(* CODESYS project tc_helper.library
   Author: R. Christopher
   Title: Tc_Helper
   Version: 1.0.0.8
   DefaultNamespace: Tc_Helper
   Company: Red Rock Controls
   Description: Clock.DateTimeInitialised added
      
      Copyright Red Rock Controls Limited 2014

Project tree, tasks and I/O mapping:
  libraries: Tc2_Standard, * (Beckhoff Automation GmbH); Tc2_System, * (Beckhoff Automation GmbH); Tc2_Utilities, * (Beckhoff Automation GmbH)
  Classes/
    function block TClock [ST]: DateAsString, DateTimeAsString, DateTimeInitialised, NowAsDateTime, NowAsTimeStruct, TimeAsString
    function block TCounter [ST]: Dec, Inc, Reset, Value, ValueAsTArg
    function block TFallingEdge [ST]: Test
    function block TOnTimer [ST]: FB_init, PresetTime, Reset, Run
    function block TRisingEdge [ST]: Test
    function block TStringSplitter [ST]: GetNext, Init
  Functions/
    function F_Concat2 [ST]
    function F_Concat4 [ST]
    function F_Concat6 [ST]
    function F_Concat8 [ST]
    function F_FormatString1 [ST]
    function F_FormatString2 [ST]
    function F_FormatString3 [ST]
    function F_FormatStringEx1 [ST]
    function F_FormatStringEx2 [ST]
    function F_FormatStringEx3 [ST]
    function F_FormatStringEx4 [ST]
    function F_LREAL_TO_STRING [ST]
    function F_LTrimEx [ST]
    function F_StripLF [ST]
    function F_Trim [ST]
    function F_UDINT_TO_STRING [ST]
  Version/
    global variables Global_Version
*)

// Version/Global_Version
// This function has been automatically generated from the project information.
VAR_GLOBAL CONSTANT
	{attribute 'const_non_replaced'}
	stLibVersion_Tc_Helper : ST_LibVersion := (iMajor := 1, iMinor := 0, iBuild := 0, iRevision := 8, sVersion := '1.0.0.8');
END_VAR

// Classes/TClock
FUNCTION_BLOCK TClock
VAR
    _DateTimeInitialised : BOOL; // to detect startup
	_NowAsTimeStruct: TIMESTRUCT;
    
	NT_GetTime1: NT_GetTime;
	TON1: TON;
    GetWindowsTimeRequest : BOOL;
	SyncRequest: BOOL;
    F_TRIG1 : F_TRIG;
	RTC_EX2: RTC_EX2;
	PresetTime: TIMESTRUCT;
END_VAR

// Request a sync every 10s
TON1(IN := NOT GetWindowsTimeRequest, PT := T#10S, Q=> GetWindowsTimeRequest);

// Get time from Windows clock
NT_GetTime1(
	NetId := '',
	Start := GetWindowsTimeRequest OR NOT _DateTimeInitialised, // request on first scan also
	TmOut := T#2S,
    Busy => ,
    Err => ,
    ErrId => ,
	TimeStr => PresetTime);

// Request sync to Windows time when time received
F_TRIG1(CLK :=  NT_GetTime1.Busy, Q=> SyncRequest);   
    
// Sync RTC to Windows time
RTC_EX2(
	EN:= SyncRequest, // re-initialise to Windows clock following sync request
	PDT:= PresetTime, // time to sync to
	PMICRO:= PresetTime.wMilliseconds, 
	Q=> , 
	CDT=> _NowAsTimeStruct, // time updated on every call
	CMICRO=> );
IF SyncRequest THEN    
    _DateTimeInitialised := TRUE;
END_IF

PROPERTY DateAsString : STRING
GET
VAR
	FB_FormatString1 : FB_FormatString;
END_VAR
FB_FormatString1(
	sFormat:= '%.2d/%.2d/%.2d', 
	arg1:= F_WORD(_NowAsTimeStruct.wDay), 
	arg2:= F_WORD(_NowAsTimeStruct.wMonth), 
	arg3:= F_WORD(_NowAsTimeStruct.wYear),
	arg4:= ,
	arg5:= , 
	arg6:= , 
	arg7:= , 
	arg8:= , 
	arg9:= , 
	arg10:= , 
	bError=> , 
	nErrId=> , 
	sOut=> DateAsString);
END_GET
END_PROPERTY

PROPERTY DateTimeAsString : STRING
GET
DateTimeAsString := F_Concat4(S1 := TimeAsString,
                              S2 := ' ',
                              S3 := DateAsString,
                              S4 := '');
END_GET
END_PROPERTY

PROPERTY DateTimeInitialised : BOOL
GET
DateTimeInitialised := _DateTimeInitialised;
END_GET
END_PROPERTY

PROPERTY NowAsDateTime : DT
GET
NowAsDateTime := SYSTEMTIME_TO_DT(TIMESTR:= _NowAsTimeStruct);
END_GET
END_PROPERTY

PROPERTY NowAsTimeStruct : TIMESTRUCT
GET
NowAsTimeStruct := _NowAsTimeStruct;
END_GET
END_PROPERTY

PROPERTY TimeAsString : STRING
GET
VAR
	FB_FormatString1 : FB_FormatString;
END_VAR
FB_FormatString1(
	sFormat:= '%.2d:%.2d:%.2d', 
	arg1:= F_WORD(_NowAsTimeStruct.wHour), 
	arg2:= F_WORD(_NowAsTimeStruct.wMinute), 
	arg3:= F_WORD(_NowAsTimeStruct.wSecond),
	arg4:= ,
	arg5:= , 
	arg6:= , 
	arg7:= , 
	arg8:= , 
	arg9:= , 
	arg10:= , 
	bError=> , 
	nErrId=> , 
	sOut=> TimeAsString);
END_GET
END_PROPERTY

END_FUNCTION_BLOCK

// Functions/F_Concat4
FUNCTION F_Concat4 : T_MaxString
VAR_INPUT
	S1: T_MaxString;
	S2: T_MaxString;
	S3: T_MaxString;
	S4: T_MaxString;
END_VAR
VAR
	Result: T_MaxString;
END_VAR

Result := CONCAT(S1,S2);
Result := CONCAT(Result,S3);
Result := CONCAT(Result,S4);
F_Concat4 := Result;

END_FUNCTION

// Classes/TCounter
FUNCTION_BLOCK TCounter
VAR
    Count : DINT;
END_VAR

METHOD Dec : DINT
VAR_INPUT
END_VAR
Count := Count - 1;
Dec := Count;
END_METHOD

METHOD Inc : DINT
VAR_INPUT
END_VAR
Count := Count + 1;
Inc := Count;
END_METHOD

METHOD Reset
VAR_INPUT
END_VAR
Count := 0;
END_METHOD

PROPERTY Value : DINT
GET
Value := Count;
END_GET
SET
Count := Value;
END_SET
END_PROPERTY

PROPERTY ValueAsTArg : T_Arg
GET
ValueAsTArg := F_DINT(Count);
END_GET
END_PROPERTY

END_FUNCTION_BLOCK

// Classes/TFallingEdge
FUNCTION_BLOCK TFallingEdge
VAR
    F_TRIG1 : F_TRIG;
END_VAR

METHOD Test : BOOL
VAR_INPUT
    Value : BOOL;
END_VAR
F_TRIG1(CLK := Value);
Test := F_TRIG1.Q;
END_METHOD

END_FUNCTION_BLOCK

// Classes/TOnTimer
FUNCTION_BLOCK TOnTimer
VAR
    TON1 : TON;
END_VAR

METHOD FB_init : BOOL
VAR_INPUT
	bInitRetains : BOOL; // if TRUE, the retain variables are initialized (warm start / cold start)
	bInCopyCode : BOOL;  // if TRUE, the instance afterwards gets moved into the copy code (online change)
    PresetTime : LREAL; // seconds
END_VAR
TON1.PT := LREAL_TO_TIME(PresetTime * 1000);
END_METHOD

PROPERTY PresetTime : LREAL
GET
PresetTime := TIME_TO_LREAL(TON1.PT)/1000.0; // in seconds
END_GET
SET
TON1.PT := LREAL_TO_TIME(PresetTime * 1000);
END_SET
END_PROPERTY

METHOD Reset
TON1(IN := FALSE);
END_METHOD

METHOD Run : BOOL
TON1(IN := TRUE);
Run := TON1.Q;
END_METHOD

END_FUNCTION_BLOCK

// Classes/TRisingEdge
FUNCTION_BLOCK TRisingEdge
VAR
    R_TRIG1 : R_TRIG;
END_VAR

METHOD Test : BOOL
VAR_INPUT
    Value : BOOL;
END_VAR
R_TRIG1(CLK := Value);
Test := R_TRIG1.Q;
END_METHOD

END_FUNCTION_BLOCK

// Classes/TStringSplitter
FUNCTION_BLOCK TStringSplitter
VAR
	SubjectString : TC2_SYSTEM.T_MaxString;
	Delimiter : STRING;
	NextDelimiterPosition : INT;
END_VAR

METHOD GetNext : STRING(255)
VAR_INPUT
END_VAR
VAR
	RemainingLength: INT;
END_VAR
NextDelimiterPosition := FIND(SubjectString , Delimiter);

IF NextDelimiterPosition > 0 THEN // delimitter found
    
    // extract next sub-string
	GetNext := LEFT(SubjectString,NextDelimiterPosition - 1);
    
    // remove sub-string from subject string
	RemainingLength := LEN(SubjectString) - NextDelimiterPosition - LEN(Delimiter) + 1;
	SubjectString := RIGHT(SubjectString,RemainingLength);
    
    // strip any delimitters from front of remaining string
    WHILE LEFT(SubjectString,1) = Delimiter DO
        SubjectString := RIGHT(SubjectString,LEN(SubjectString) - 1);
	END_WHILE
ELSE
	GetNext := SubjectString; // return what is left
	SubjectString := '';
END_IF
END_METHOD

METHOD Init
VAR_INPUT
		Str : TC2_SYSTEM.T_MaxString;
		Delim : STRING;
END_VAR
SubjectString := Str;
NextDelimiterPosition := 0;
Delimiter := Delim;
END_METHOD

END_FUNCTION_BLOCK

// Functions/F_Concat2
FUNCTION F_Concat2 : T_MaxString
VAR_INPUT
	S1: T_MaxString;
	S2: T_MaxString;
END_VAR
VAR
	Result: T_MaxString;
END_VAR

Result := CONCAT(S1,S2);
F_Concat2 := Result;

END_FUNCTION

// Functions/F_Concat6
FUNCTION F_Concat6 : T_MaxString
VAR_INPUT
	S1: T_MaxString;
	S2: T_MaxString;
	S3: T_MaxString;
	S4: T_MaxString;
	S5: T_MaxString;
	S6: T_MaxString;
END_VAR
VAR
	Result: T_MaxString;
END_VAR

Result := CONCAT(S1,S2);
Result := CONCAT(Result,S3);
Result := CONCAT(Result,S4);
Result := CONCAT(Result,S5);
Result := CONCAT(Result,S6);
F_Concat6 := Result;

END_FUNCTION

// Functions/F_Concat8
FUNCTION F_Concat8 : T_MaxString
VAR_INPUT
	S1: T_MaxString;
	S2: T_MaxString;
	S3: T_MaxString;
	S4: T_MaxString;
	S5: T_MaxString;
	S6: T_MaxString;
	S7: T_MaxString;
	S8: T_MaxString;
END_VAR
VAR
	Result: T_MaxString;
END_VAR

Result := CONCAT(S1,S2);
Result := CONCAT(Result,S3);
Result := CONCAT(Result,S4);
Result := CONCAT(Result,S5);
Result := CONCAT(Result,S6);
Result := CONCAT(Result,S7);
Result := CONCAT(Result,S8);
F_Concat8 := Result;

END_FUNCTION

// Functions/F_FormatString1
FUNCTION F_FormatString1 : T_MaxString
VAR_INPUT
	Format	: T_MaxString;
	arg1	: T_Arg;
END_VAR
VAR
    FB_FormatString1 : FB_FormatString;
END_VAR

FB_FormatString1(
	sFormat:= Format, 
	arg1:= arg1, 
	arg2:= , 
	arg3:= , 
	arg4:= , 
	arg5:= , 
	arg6:= , 
	arg7:= , 
	arg8:= , 
	arg9:= , 
	arg10:= , 
	bError=> , 
	nErrId=> , 
	sOut=> F_FormatString1);

END_FUNCTION

// Functions/F_FormatString2
FUNCTION F_FormatString2 : T_MaxString
VAR_INPUT
	Format	: T_MaxString;
	arg1	: T_Arg;
	arg2	: T_Arg;
END_VAR
VAR
    FB_FormatString1 : FB_FormatString;
END_VAR

FB_FormatString1(
	sFormat:= Format, 
	arg1:= arg1, 
	arg2:= arg2, 
	arg3:= , 
	arg4:= , 
	arg5:= , 
	arg6:= , 
	arg7:= , 
	arg8:= , 
	arg9:= , 
	arg10:= , 
	bError=> , 
	nErrId=> , 
	sOut=> F_FormatString2);

END_FUNCTION

// Functions/F_FormatString3
FUNCTION F_FormatString3 : T_MaxString
VAR_INPUT
	Format	: T_MaxString;
	arg1	: T_Arg;
	arg2	: T_Arg;
	arg3	: T_Arg;
END_VAR
VAR
    FB_FormatString1 : FB_FormatString;
END_VAR

FB_FormatString1(
	sFormat:= Format, 
	arg1:= arg1, 
	arg2:= arg2, 
	arg3:= arg3, 
	arg4:= , 
	arg5:= , 
	arg6:= , 
	arg7:= , 
	arg8:= , 
	arg9:= , 
	arg10:= , 
	bError=> , 
	nErrId=> , 
	sOut=> F_FormatString3);

END_FUNCTION

// Functions/F_FormatStringEx1
FUNCTION F_FormatStringEx1 : T_MaxString
VAR_INPUT
	Format	: T_MaxString;
	arg1	: T_MaxString;
END_VAR
VAR
    FB_FormatString1 : FB_FormatString;
END_VAR



FB_FormatString1(
	sFormat:= Format, 
	arg1:= F_STRING(arg1), 
	arg2:= , 
	arg3:= , 
	arg4:= , 
	arg5:= , 
	arg6:= , 
	arg7:= , 
	arg8:= , 
	arg9:= , 
	arg10:= , 
	bError=> , 
	nErrId=> , 
	sOut=> F_FormatStringEx1);

END_FUNCTION

// Functions/F_FormatStringEx2
FUNCTION F_FormatStringEx2 : T_MaxString
VAR_INPUT
	Format	: T_MaxString;
	arg1	: T_MaxString;
	arg2	: T_MaxString;
END_VAR
VAR
    FB_FormatString1 : FB_FormatString;
END_VAR



FB_FormatString1(
	sFormat:= Format, 
	arg1:= F_STRING(arg1), 
	arg2:= F_STRING(arg2),
	arg3:= , 
	arg4:= , 
	arg5:= , 
	arg6:= , 
	arg7:= , 
	arg8:= , 
	arg9:= , 
	arg10:= , 
	bError=> , 
	nErrId=> , 
	sOut=> F_FormatStringEx2);

END_FUNCTION

// Functions/F_FormatStringEx3
FUNCTION F_FormatStringEx3 : T_MaxString
VAR_INPUT
	Format	: T_MaxString;
	arg1	: T_MaxString;
	arg2	: T_MaxString;
	arg3	: T_MaxString;
END_VAR
VAR
    FB_FormatString1 : FB_FormatString;
END_VAR



FB_FormatString1(
	sFormat:= Format, 
	arg1:= F_STRING(arg1), 
	arg2:= F_STRING(arg2),
	arg3:= F_STRING(arg3), 
	arg4:= , 
	arg5:= , 
	arg6:= , 
	arg7:= , 
	arg8:= , 
	arg9:= , 
	arg10:= , 
	bError=> , 
	nErrId=> , 
	sOut=> F_FormatStringEx3);

END_FUNCTION

// Functions/F_FormatStringEx4
FUNCTION F_FormatStringEx4 : T_MaxString
VAR_INPUT
	Format	: T_MaxString;
	arg1	: T_MaxString;
	arg2	: T_MaxString;
	arg3	: T_MaxString;
	arg4	: T_MaxString;
END_VAR
VAR
    FB_FormatString1 : FB_FormatString;
END_VAR



FB_FormatString1(
	sFormat:= Format, 
	arg1:= F_STRING(arg1), 
	arg2:= F_STRING(arg2),
	arg3:= F_STRING(arg3), 
	arg4:= F_STRING(arg4), 
	arg5:= , 
	arg6:= , 
	arg7:= , 
	arg8:= , 
	arg9:= , 
	arg10:= , 
	bError=> , 
	nErrId=> , 
	sOut=> F_FormatStringEx4);

END_FUNCTION

// Functions/F_LREAL_TO_STRING
FUNCTION F_LREAL_TO_STRING : STRING
VAR_INPUT
    Value : LREAL;
    Precision : INT;
END_VAR
VAR
END_VAR

F_LREAL_TO_STRING := LREAL_TO_FMTSTR(in := Value,
                                     iPrecision := Precision,
                                     bRound := TRUE);

END_FUNCTION

// Functions/F_LTrimEx
FUNCTION F_LTrimEx : T_MaxString // removes n characters from start of string
VAR_INPUT
   n : UINT; 
   str : T_MaxString;
END_VAR
VAR
    Length : UINT;
END_VAR

Length := INT_TO_UINT(LEN(str));
IF n = 0 THEN
    F_LTrimEx := str;
ELSIF n < Length THEN
    MEMCPY(destAddr := ADR(F_LTrimEx),
           srcAddr  := ADR(str) + n,
           n        := Length - n + 1); // include null terminator
END_IF

END_FUNCTION

// Functions/F_StripLF
FUNCTION F_StripLF : T_MaxString
VAR_INPUT
    str : STRING;
END_VAR
VAR
    pChar : POINTER TO BYTE;
    i : INT;
END_VAR

pChar := ADR(str);
FOR i := 0 TO LEN(Str)-1 DO
    IF pChar[i] = 16#0D OR pChar[i] = 16#0A THEN
        pChar[i] := 0;
	END_IF
END_FOR
F_StripLF := str;

END_FUNCTION

// Functions/F_Trim
FUNCTION F_Trim : T_MaxString
VAR_INPUT
	in: T_MaxString;
END_VAR
VAR
	Result: T_MaxString;
END_VAR

Result := F_LTrim(F_RTrim(In));
WHILE LEFT(Result,1) = '$T' DO
	Result := RIGHT(Result,LEN(Result)-1); // Strip tabs,too
END_WHILE
F_Trim := Result;

END_FUNCTION

// Functions/F_UDINT_TO_STRING
FUNCTION F_UDINT_TO_STRING : STRING
VAR_INPUT
    Value : UDINT;
END_VAR
VAR
END_VAR

F_UDINT_TO_STRING := DWORD_TO_HEXSTR(Value,4,FALSE);

END_FUNCTION
